FUNCTION CIRCLE_A : REAL
VAR_INPUT
	rx : REAL;
	ax : REAL;
END_VAR


(*
version 1.2	22. feb 2008
programmer 	hugo
tested by		tobias

circle_A calculates the Area of a circle segement if ax = 360 the whole circle is calculated


*)

circle_A := Rx * RX * 8.726646E-3 * Ax;

(* revision histroy
hm	16. oct 2007	rev 1.0
	original version

hm	4. dec 2007		rev 1.1
	changed code for better performance

hm	22. feb 2008	rev 1.2
	improved performance
*)

END_FUNCTION

(* stored: Version 1.1.0.1, ProductVersion 3.1.4022.7
   POU CIRCLE_A: Id {3a6291e1-5144-4470-bebb-c1065423220a}, SpecialFunc None *)
